{attribute 'linkalways'} 
{attribute 'no_explicit_call' := 'This FB is a CLASS and must be accessed using methods or properties'}
{attribute 'enable_dynamic_creation'}
FUNCTION_BLOCK Node_F_VN_ResizeImage EXTENDS VisionNode
VAR
    ipSrcImage : _ITcVnImage;
    ipDestImage : _ITcVnImage;
    nWidth : _UDINT(0);
    nHeight : _UDINT(0);
    eInterpolationType : _ETcVnInterpolationType(ETcVnInterpolationType.TCVN_IT_NEAREST_NEIGHBOR);
    hrPrev : _HRESULT(S_OK);
	hresult : _HRESULT(S_OK);
END_VAR

METHOD PUBLIC  Clone : I_Node
VAR
	pNode : POINTER TO Node_F_VN_ResizeImage;
END_VAR
pNode := __NEW(Node_F_VN_ResizeImage);
Clone := pNode^;
END_METHOD

METHOD FB_init : BOOL
VAR_INPUT
	bInitRetains : BOOL; // if TRUE, the retain variables are initialized (warm start / cold start)
	bInCopyCode : BOOL;  // if TRUE, the instance afterwards gets moved into the copy code (online change)
END_VAR
AddInput('ipSrcImage', ipSrcImage);
AddInput('nWidth', nWidth);
AddInput('nHeight', nHeight);
AddParameter('eInterpolationType', eInterpolationType);
AddInput('hrPrev', hrPrev);
AddOutput('ipDestImage', ipDestImage);
AddOutput('hresult',hresult);
END_METHOD

METHOD PROTECTED OnExecute
hresult.Value := F_VN_ResizeImage(
    ipSrcImage := ipSrcImage.Value,
	ipDestImage := ipDestImage.Value,
    nWidth := nWidth.Value,
    nHeight := nHeight.Value,
    eInterpolationType := eInterpolationType.Value,
	hrPrev:= hrPrev.Value);
END_METHOD

METHOD PUBLIC PreExecutionCheck
VAR_INPUT
	Check : I_PreExecutionChecks;
END_VAR
Check.IsTrue(ipSrcImage.IsValid, 'ipSrcImage must contain an image');
END_METHOD

END_FUNCTION_BLOCK

(* stored: Version 1.1.0.1, ProductVersion 3.1.4024.13
   POU Node_F_VN_ResizeImage: Id {0721970a-3821-0d06-364e-a85f8b044a3d}, SpecialFunc None
   Folder Constructor: Id {28106f39-b343-0cc6-1145-7dda6b5cac17}
   Method Clone: Id {de747080-9729-09aa-3225-7dcfa513bc3b}
   Method FB_init: Id {df441881-747c-0ff1-2c5e-01c547fb8c1b}
   Method OnExecute: Id {3afb66cf-1262-0e82-3d3e-9db9b7e4c3c5}
   Method PreExecutionCheck: Id {29a3c58c-dd81-0188-329f-8ff8ab5e4abf} *)
